// TIA Portal V16 export
// export: Created 2025-05-30T16:30:45.4613706Z, ExportSetting WithDefaults, DisplayName Totally Integrated Automation Portal, DisplayVersion V16, DisplayName TIA Portal Version Control Interface, DisplayVersion V16, DisplayName TIA Portal Openness, DisplayVersion V16, DisplayName STEP 7 Professional, DisplayVersion V16, DisplayName STEP 7 Safety, DisplayVersion V16, DisplayName WinCC Advanced, DisplayVersion V16
DATA_BLOCK "Alarm_Axis_Position_Function_Wals"   // DB41
VERSION : 0.1
// stored: AutoNumber true, InstanceOfName Alarm_Axis_Position_Function, InstanceOfType FB
"Alarm_Axis_Position_Function"
   // VAR_INPUT
   //    "Axis FWD command" : Bool;
   //    "Axis Feedback (Sensor) signal" : Bool;
   //    "Axis Encoder Singal" : Real;
   //    "Axis Command Position" : Real;
   //    "Sensor Controlled (HIGH) - Position Controlled (LOW)" : Bool;
   //    "CheckTime Setting" : Time;
   // END_VAR
   // VAR_OUTPUT
   //    "Alarm BOOL" : Bool;
   //    "Alarm WORD" : Bool;
   // END_VAR
BEGIN
END_DATA_BLOCK
